(* IEC 61131-3 sources: Controls/Draft codes/Structured Text, 4 files *)

(* ---- emergency_shutdown.st ---- *)
// Assumptions
    // the emergency shutdown state is triggered only if SYSTEM_FAIL is TRUE
	// the variable SYSTEM_FAIL will be passed into the function
	// currentState represents the state the system is currently in
PROGRAM	 emergency_shutdown
	FUNCTION check_shutdown
		VAR_INPUT
        	system_fail: BOOL;
		END_VAR
		IF system_fail
			IF POD_ACCELERATION > 0
				// close propulsion valves (subroutine)
				closePropValves();
			// activate brakes (subroutine)
			activateBrake();

			IF PROP_TNK_PRES != 0
				// Release Remaining pressure Tank (subroutine)
				releasePressure();

			// trigger stop state (set currentState to stop
			currentState = -1;
			// -1 is a placeholder, replace with corresponding enum val
	END_FUNCTION

	FUNCTION activateBrake
		// set brake pins to on
		// Brake pins (NOV-1, NOV-2, NOV-3, NOV-4, NCV-1, NCV-2)
		// are set to 0
	END_FUNCTION

	FUNCTION releasePressure
		// set pressure pins to on
	END_FUNCTION

	FUNCTION closePropValves
		// set S-1, S-2, S-3, S-4 to 0
	END_FUNCTION

END_PROGRAM

(* ---- emergencyshutdown.st ---- *)
PROGRAM Emergency_Shutdown
    FUNCTION CheckShutdown
        VAR_INPUT
            system_fail: BOOL;
        END_VAR
        VAR
            pod_accelaration: INT;
            tank_pressure: INT;
        END_VAR
        IF system_fail THEN
            pod_accelaration := GETPODACCELARATION();
            IF pod_accelaration > 0 THEN
                ClosePropValves();
            END_IF
            ActivateBrake();
            IF tank_pressure <> 0 THEN
                ReleasePressure();
            END_IF
            CURRENT_STATE = -1;
        END_IF
    END_FUNCTION
    FUNCTION ActivateBrake

    END_FUNCTION
    FUNCTION ReleasePressure

    END_FUNCTION
    FUNCTION ClosePropValves

    END_FUNCTION
END_PROGRAM

(* ---- state_updater.st ---- *)
PROGRAM update_states
    /*
    cmd = 1 -> BEGIN cmd  M
    cmd = 2 -> IDLE    M
    cmd = 3 -> ARM     M
    cmd = 4 -> LAUNCH  M
    cmd = 5 -> stop  A/M
    cmd = 6 -> CRAWL M
    cmd = 7 -> END   M
    cmd = 8 -> EGSD  A/M
    cmd = 9 -> coast A

    1  idle
    2  System check
    3  Armed
    4  Acceleration
    5  Coast
    6  Brake
    7  stop
    8  CRAWL
    9  End
    10 Emergency shutdown
    */
    VAR_INPUT
        currState: INT;
        cmd: INT;
        END_VAR
        VAR_OUTPUT
            newState: INT;

    VAR
        newState: INT = 0;
    END_VAR

    FUNCTION update
        // go to emergency shutdown
        IF cmd == 8 THEN
            newState = 10;

        //transiton 1
        IF cmd ==2 && currState == 1 THEN
            newState =2;

        // transition 2
        IF cmd ==1 && currState ==2 THEN
            newState = 1;

        // transition 3
        IF cmd == 3 && currState == 2 THEN
            newState = 3;

        // transition 4
        IF cmd == 4 && currState == 3 THEN
            newState = 4;

        // transition 5
        IF currState == 4 && cmd == 9 THEN
            newState = 5;

        // transition 6
        IF currState == 5 && cmd == 5 THEN
            newState = 6;

        // transition 7
        IF currState == 6 && POD_VELOCITY <= 0 THEN
            newState = 7;

        // transition 8
        IF currState == 7 && cmd == 6 THEN
            newState = 8;

        // transition 9
        IF currState == 8 && cmd == 5 THEN
            newState = 6;

        // transition 10
        IF currState == 7 && cmd == 7 THEN
            newState = 9;
    END_FUNCTION
END_PROGRAM

(* ---- triggershutdown.st ---- *)
PROGRAM Trigger_Shutdown
    FUNCTION Trigger
        VAR_INPUT

        END_VAR
        VAR_OUTPUT
            system_fail: BOOL;
        END_VAR
        VAR
            brake_eval_int: INT;
            brake_eval_bool: BOOL;
            prop_eval_bool: BOOL;
            bat_eval_bool: BOOL;
            comm_eval_bool: BOOL;
        END_VAR
        EvalBrake(brake_eval_int);
        IF brake_eval_int >= 2 THEN
            brake_eval_bool := FALSE;
            system_fail := TRUE;
            EvalProp(prop_eval_bool);
        ELSE IF NOT(prop_eval_bool) THEN
            prop_eval_bool := FALSE;
            system_fail := TRUE;
            EvalBattery(bat_eval_bool);
        ELSE IF NOT(prop_eval_bool) THEN
            bat_eval_bool := FALSE;
            system_fail := TRUE;
            EvalComm(comm_eval_bool);
        ELSE IF NOT(comm_eval_bool) THEN
            comm_eval_bool := FALSE;
            system_fail := TRUE;
        ELSE THEN
            system_fail := FALSE;
        END_IF
    END_FUNCTION
    FUNCTION EvalBrake
        VAR_INPUT

        END_VAR
        VAR_OUTPUT
            brake_state: INT;
        END_VAR
        brake_state := BRAKE_SUBSTATE1 + BRAKE_SUBSTATE2;
    END_FUNCTION
    FUNCTION EvalProp
        VAR_INPUT

        END_VAR
        VAR_OUTPUT
            prop_state: BOOL;
        END_VAR
        prop_state := PROP_STATE;
    END_FUNCTION
    FUNCTION EvalBattery
        VAR_INPUT

        END_VAR
        VAR_OUTPUT
            batt_state: BOOL;
        END_VAR
        batt_state := BATT_STATE;
    END_FUNCTION
    FUNCTION EvalComm
        VAR_INPUT

        END_VAR
        VAR_OUTPUT
            comm_state: BOOL;
        END_VAR
        comm_state := COMM_STATE;
    END_FUNCTION
END_PROGRAM
